FUNCTION_BLOCK FB_FieldCodecFloat EXTENDS FB_FieldCodec
VAR_INPUT
END_VAR
VAR_OUTPUT
END_VAR
VAR
    fValue : REAL;
END_VAR

METHOD CalculatePackedDataSize : HRESULT
VAR_INPUT CONSTANT
	anyFirstElem	: T_Any;
	nLength	        : UDINT;        // items to write
END_VAR
VAR_OUTPUT
    nPackedDataSize : UDINT;
END_VAR
VAR
    anyItem         : T_ANY;
    i               : UDINT;
    fValue          : REAL;
END_VAR
anyItem := anyFirstElem;

IF nLength < 1 THEN
    nPackedDataSize := 0;
    RETURN;
END_IF

FOR i := 0  TO nLength - 1 DO
    anyItem.pValue := anyFirstElem.pValue + (i * TO_UDINT(anyFirstElem.diSize)); 
    fValue := PREAL_TO_REAL(anyItem.pValue);
    nPackedDataSize := nPackedDataSize + F_ComputeFloatSize(fValue);
END_FOR
END_METHOD

METHOD IsPackedRepeatedField : BOOL
VAR_INPUT
	nTag	: UDINT;
END_VAR
IsPackedRepeatedField := F_IsPackedRepeatedField(nTag);
END_METHOD


METHOD ValueReader : HRESULT
VAR_IN_OUT      
    stCtx : ST_ParseContext;
END_VAR
VAR_OUTPUT
	anyOut	: T_Any;
END_VAR

ValueReader := F_ParseFloat(stCtx, fValue=> fValue);
anyOut := F_ToAnyType(anyArg:= fValue);
END_METHOD

METHOD ValueWriter : HRESULT
VAR_IN_OUT
    stCtx  : ST_WriteContext;
END_VAR
VAR_INPUT
    anyIn : T_ANY;
END_VAR
VAR
    fValue  : REAL;
END_VAR

fValue := PREAL_TO_REAL(anyIn.pValue);
ValueWriter := F_WriteFloat(stCtx, fValue);
END_METHOD

END_FUNCTION_BLOCK

(* stored: Version 1.1.0.1
   POU FB_FieldCodecFloat: Id {456f0824-5fc9-4ac6-93a6-44622df993e1}, SpecialFunc None
   Method CalculatePackedDataSize: Id {b1448257-0eb4-4d38-9454-f8efab3d64b3}
   Method IsPackedRepeatedField: Id {67837a61-ee94-486b-b084-c1e5db16fd13}
   Method ValueReader: Id {fd6da9dd-5a95-4a2b-9b04-99f6349f20b2}
   Method ValueWriter: Id {82739368-41e6-4d6c-82cd-f15dee5abfbd} *)
